TYPE "Analogic_SensorManagement_Warning"
VERSION : 0.1
// Block: Analogic_SensorManagement_Warning
   STRUCT
      PresetNeed : Bool;
      SignalError : Bool;
      SensorDisabled : Bool;
   END_STRUCT;

END_TYPE
